// Mitsubishi GX Works2 project: 적산타이머   PLC: Q02/Q02H

PROGRAM MAIN
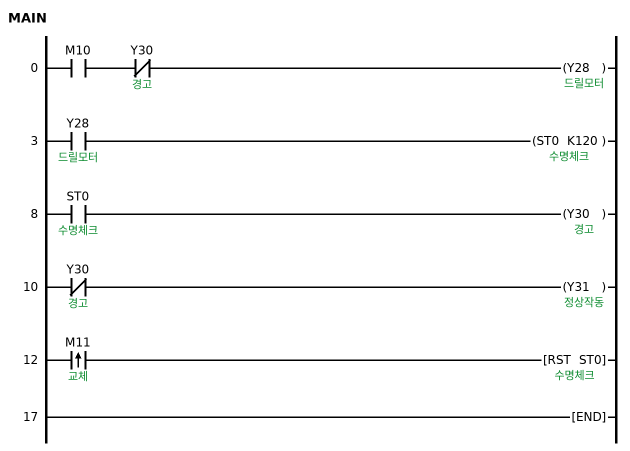
0     LD      M10
      ANI     Y30  ; 경고
      OUT     Y28  ; 드릴모터
3     LD      Y28  ; 드릴모터
      OUT     ST0 K120  ; 수명체크
8     LD      ST0  ; 수명체크
      OUT     Y30  ; 경고
10    LDI     Y30  ; 경고
      OUT     Y31  ; 정상작동
12    LDP     M11  ; 교체
      RST     ST0  ; 수명체크
17    END
END_PROGRAM
